PROGRAM P_MachineControl
VAR
	fbInverse					: FB_InverseKin2d;
	fRefPosX					: LREAL := GVL_InverseKinematics.fTooltipXCoordGlobalIni;
	fRefPosY					: LREAL := GVL_InverseKinematics.fTooltipYCoordGlobalIni;					
END_VAR

G_Work.bManualMode := G_Inputs.bManualModeSelector;
G_Work.bAutoMode := G_Inputs.bAutoModeSelector;

IF G_Inputs.bAutoModeSelector THEN
fRefPosX := fRefPosX + G_Sensors.fJoystickLeftNormalizedX*-0.001;
fRefPosY := fRefPosY + G_Sensors.fJoystickLeftNormalizedY*0.001;
END_IF

fbInverse(
	fPtXd := fRefPosX, 
	fPtYd := fRefPosY, 
	fTheta1 :=GVL_InverseKinematics.fTheta1,
	
	fTheta3 => GVL_InverseKinematics.fAngleMainArmInverse, 
	fTheta4 => GVL_InverseKinematics.fAngleKnuckleArmInverse,
	fStrokeActuatorMain => GVL_InverseKinematics.fStrokeActuatorMainInverse,
	fStrokeActuatorKnuckle => GVL_InverseKinematics.fStrokeActuatorKnuckleInverse,	
);

END_PROGRAM

(* stored: Version 1.1.0.1, ProductVersion 3.1.4024.12
   POU P_MachineControl: Id {a90e0789-57c0-407b-b2f1-afc96a165b42}, SpecialFunc None *)
